FUNCTION_BLOCK FB_VfdIOControl
VAR_INPUT
	bStartMotor			AT %Q*: BOOL;
	bStopMotor			AT %Q*: BOOL;
	nSetSpeed 			AT %Q*: INT;
	nActualSpeed		AT %I*: INT;
	bRemoteLocalStatus  AT %I* : BOOL;
END_VAR
VAR_OUTPUT
END_VAR
VAR

END_VAR

END_FUNCTION_BLOCK

(* stored: Version 1.1.0.1, ProductVersion 3.1.4024.5
   POU FB_VfdIOControl: Id {250181c0-7f7c-4abb-aa48-a0818c359bac}, SpecialFunc None *)
